{attribute 'qualified_only'}
{attribute 'strict'}
TYPE E_TuneMode :
(
	Normal := 0,
	Fast := 1,
	Slow :=2
);
END_TYPE

(* stored: Version 1.1.0.1, ProductVersion 3.1.4024.12
   DUT E_TuneMode: Id {bb478196-20bc-4d9d-bc97-c543a2506dc1} *)
